(* Logix 5000 project; controller PRJ_108_1 vendor 1 type 14 code 216 rev 34.11; software revision 34.01 *)

TASK MainTask (continuous, watchdog 500 ms) : MainProgram

MODULES
   Local : vendor 1 type 14 code 216 (5069 0, rev 34.11)
      VFD_7 : PowerFlex 525-EENET (Ethernet 192.168.1.118, rev 7.1, Output RPI 20 ms)
      VFD_8 : PowerFlex 525-EENET (Ethernet 192.168.1.119, rev 7.1, Output RPI 20 ms)
      VFD112 : vendor 1 type 142 code 1168 (Ethernet 192.168.1.112, rev 16.2, Output RPI 20 ms)
          : vendor 1 type 142 code 767 (RhinoBP 1, rev 2.7)
          : vendor 1 type 142 code 33184 (RhinoBP 14, rev 2.5)
          : vendor 1 type 142 code 57760 (RhinoBP 6, rev 1.2)
      VFD_6 : PowerFlex 525-EENET (Ethernet 192.168.1.117, rev 7.1, Output RPI 20 ms)
      VFD_4 : PowerFlex 525-EENET (Ethernet 192.168.1.115, rev 7.1, Output RPI 20 ms)
      VFD_5 : PowerFlex 525-EENET (Ethernet 192.168.1.116, rev 7.1, Output RPI 20 ms)
      VFD_9 : PowerFlex 525-EENET (Ethernet 192.168.1.120, rev 7.1, Output RPI 20 ms)
      VFD113 : vendor 1 type 142 code 1168 (Ethernet 192.168.1.113, rev 16.2, Output RPI 20 ms)
          : vendor 1 type 142 code 767 (RhinoBP 1, rev 2.7)
          : vendor 1 type 142 code 57760 (RhinoBP 6, rev 1.2)
          : vendor 1 type 142 code 33184 (RhinoBP 14, rev 2.5)
      VFD_114 : vendor 1 type 127 code 41 (Ethernet 192.168.1.114, rev 8.2, Output RPI 20 ms)
          : vendor 1 type 127 code 33792 (DSI 1, rev 1.9)
      NODE_1 : 1734-AENT (Ethernet 192.168.1.111, rev 6.1, Output RPI 20 ms)
         N1S11 : 1734-IB8 (PointIO 11, rev 3.1)
         N1S1 : 1734-IB8 (PointIO 1, rev 3.1)
         N1S10 : 1734-IB8 (PointIO 10, rev 3.1)
         N1S13 : 1734-IB8 (PointIO 13, rev 3.1)
         N1S14 : 1734-IB8 (PointIO 14, rev 3.1)
         N1S5 : 1734-IB8 (PointIO 5, rev 3.1)
         N1S3 : 1734-IB8 (PointIO 3, rev 3.1)
         N1S9 : 1734-IB8 (PointIO 9, rev 3.1)
         N1S2 : 1734-IB8 (PointIO 2, rev 3.1)
         N1S33 : vendor 1 type 115 code 210 (PointIO 33, rev 3.1, Input RPI 80 ms)
         N1S31 : vendor 1 type 115 code 210 (PointIO 31, rev 3.1, Input RPI 80 ms)
         N1S16 : 1734-IB8 (PointIO 16, rev 3.1)
         N1S19 : 1734-IB8 (PointIO 19, rev 3.1)
         N1S12 : 1734-IB8 (PointIO 12, rev 3.1)
         N1S15 : 1734-IB8 (PointIO 15, rev 3.1)
         N1S20 : 1734-IB8 (PointIO 20, rev 3.1)
         N1S6 : 1734-IB8 (PointIO 6, rev 3.1)
         N1S7 : 1734-IB8 (PointIO 7, rev 3.1)
         N1S32 : vendor 1 type 115 code 210 (PointIO 32, rev 3.1, Input RPI 80 ms)
         N1S4 : 1734-IB8 (PointIO 4, rev 3.1)
         N1S18 : 1734-IB8 (PointIO 18, rev 3.1)
         N1S8 : 1734-IB8 (PointIO 8, rev 3.1)
         N1S17 : 1734-IB8 (PointIO 17, rev 3.1)
         N1S30 : 1734-OB8 (PointIO 30, rev 3.1)
         N1S34 : vendor 1 type 115 code 211 (PointIO 34, rev 3.1, Output RPI 80 ms)
         N1S28 : 1734-OB8 (PointIO 28, rev 3.1)
         N1S22 : 1734-OB8 (PointIO 22, rev 3.1)
         N1S21 : 1734-OB8 (PointIO 21, rev 3.1)
         N1S24 : 1734-OB8 (PointIO 24, rev 3.1)
         N1S29 : 1734-OB8 (PointIO 29, rev 3.1)
         N1S35 : 1734-OE2C (PointIO 35, rev 3.1, Output RPI 80 ms)
         N1S27 : 1734-OB8 (PointIO 27, rev 3.1)
         N1S23 : 1734-OB8 (PointIO 23, rev 3.1)
         N1S26 : 1734-OB8 (PointIO 26, rev 3.1)
         N1S25 : 1734-OB8 (PointIO 25, rev 3.1)
END_MODULES

PROGRAM MainProgram   (* main routine MainRoutine *)

ROUTINE MainRoutine   (* ladder *)
END_ROUTINE
END_PROGRAM
